{attribute 'GeneratedUsingTerminal: EP2816-0008-0018'}
{attribute addProperty BoxType "EP2816-0008-0018"}
{attribute addProperty Id "OutputAT %Q*ARRAY[0..7] OF BOOL8"}
{attribute addProperty CRC "1253840710"}
{attribute addProperty Size "8"}
TYPE DIG_Outputs_Channel_28AC1A9E EXTENDS OutputBase_10CEE7DE :
STRUCT
	{attribute addProperty Name "Output"}
	Output AT %Q* : ARRAY[0..7] OF BOOL;
END_STRUCT
END_TYPE

(* stored: Version 1.2.0.0, ProductVersion 3.1.4024.11
   DUT DIG_Outputs_Channel_28AC1A9E: Id {07f360db-0e18-4a0b-904f-37521489463a} *)
